// TwinCAT 3 PLC project Untitled1
// ProgramVersion: 3.1.4022.7
// libraries:
//   Tc2_MC2, * (Beckhoff Automation GmbH)
//   Tc2_MC2_Camming, * (Beckhoff Automation GmbH)
//   Tc2_Standard, * (Beckhoff Automation GmbH)
//   Tc2_System, * (Beckhoff Automation GmbH)
//   Tc3_Module, * (Beckhoff Automation GmbH)
// project tree:
//   DUTs/ ST_AxisIN.TcDUT, ST_AxisInterface.TcDUT, ST_AxisOUT.TcDUT
//   GVLs/ GVL_Servo.TcGVL
//   / PlcTask.TcTTO
//   POUs/ FB_Servo.TcPOU, MAIN.TcPOU, PRG_Camming.TcPOU
// real-time tasks:
//   TASK PlcTask: cycle T#10ms, priority 20, ADS port 350
// motion (NC):
//   TASK NC-Task 1 SAF: cycle T#2ms, priority 4, ADS port 501
//   TASK NC-Task 1 SVB: cycle T#10ms, priority 8, ADS port 511
//   AXIS Axis 3 (id 3)
//     Dynamic: Acceleration=12830, Deceleration=12830, Jerk=38490
//     Velo: RefSearch=85, RefSync=85, SlowManual=427, FastManual=2566, Fast=8553, Maximum=8553
//     OtherSettings: AllowMotionCmdToSlave=true
//     encoder EncType=8
//       EncPara: ScaleFactorNumerator=100, ScaleFactorDenominator=1048576, MaxCount=#xffffffff
//     drive DrvType=9
//       DrvPara: MaxCount=#xffffffff, DriveControlDWord=#x00030100
//         Analog: VeloReferenz=9408, ScaleFactorActTorque=0.1
//         TimeComp: TaskDelayCycles=1
//     controller CtrType=1
//       CtrPara: PriorControlFactor=1
//         Observer: BandWidth=20
//   AXIS Axis 4 (id 4)
//     Dynamic: Acceleration=12632, Deceleration=12632, Jerk=37898
//     Velo: RefSearch=84, RefSync=84, SlowManual=421, FastManual=2526, Fast=8421, Maximum=8421
//     OtherSettings: AllowMotionCmdToSlave=true
//     encoder EncType=8
//       EncPara: ScaleFactorNumerator=100, ScaleFactorDenominator=1048576, MaxCount=#xffffffff
//     drive DrvType=9
//       DrvPara: MaxCount=#xffffffff, DriveControlDWord=#x00030100
//         Analog: VeloReferenz=9264, ScaleFactorActTorque=0.1
//         TimeComp: TaskDelayCycles=1
//     controller CtrType=1
//       CtrPara: PriorControlFactor=1
//         Observer: BandWidth=20
// I/O:
//   DEVICE Device 1 (EtherCAT), AmsNetId 192.168.2.60.2.1
//     Term 1 (EK1200) [EK1200-5000 EtherCAT Power supply (2A E-Bus)]
//       Term 2 (EL1004) [EL1004 4Ch. Dig. Input 24V, 3ms]
//       Term 3 (EL2004) [EL2004 4Ch. Dig. Output 24V, 0.5A]
//       Term 4 (EL3062) [EL3062 2Ch. Ana. Input 0-10V]
//       Term 5 (EL4002) [EL4002 2Ch. Ana. Output 0-10V, 12bit]
//       Term 6 (EK1110) [EK1110 EtherCAT extension]
//     Drive 7 (AX5203-0000-0203) [AX5203-0000-0203 EtherCAT Drive (SoE, 2 Ch.)]
//   DEVICE Device 4 (USB)
//     Box 1 (CX2100 Power Supply)
//   DEVICE Device 5 (NOV-DP-RAM)
// variable links:
//   NC-Task 1 SAF/Axes/Axis 3 <-> Device 1 (EtherCAT)/Drive 7 (AX5203-0000-0203)
//     Drive/Inputs/In/nDataIn1 <-> AT 1/Following distance
//     Drive/Inputs/In/nDcOutputTime <-> InfoData/DcOutputShift
//     Drive/Inputs/In/nState1 <-> AT 1/Drive status word @bit 8
//     Drive/Inputs/In/nState2 <-> AT 1/Drive status word
//     Drive/Inputs/In/nState4 @bit 1 <-> WcState/InputToggle
//     Drive/Inputs/In/nState4 <-> WcState/WcState
//     Drive/Outputs/Out/nCtrl1 <-> MDT 1/Master control word @bit 8
//     Drive/Outputs/Out/nDataOut1 <-> MDT 1/Position command value
//     Enc/Inputs/In/nDataIn1 <-> AT 1/Position feedback 1 value
//     Enc/Inputs/In/nDcInputTime <-> InfoData/DcInputShift
//     Enc/Inputs/In/nState4 @bit 1 <-> WcState/InputToggle
//     Enc/Inputs/In/nState4 <-> WcState/WcState
//   NC-Task 1 SAF/Axes/Axis 4 <-> Device 1 (EtherCAT)/Drive 7 (AX5203-0000-0203)
//     Drive/Inputs/In/nDataIn1 <-> AT 2/Following distance
//     Drive/Inputs/In/nDcOutputTime <-> InfoData/DcOutputShift
//     Drive/Inputs/In/nState1 <-> AT 2/Drive status word @bit 8
//     Drive/Inputs/In/nState2 <-> AT 2/Drive status word
//     Drive/Inputs/In/nState4 @bit 1 <-> WcState/InputToggle
//     Drive/Inputs/In/nState4 <-> WcState/WcState
//     Drive/Outputs/Out/nCtrl1 <-> MDT 2/Master control word @bit 8
//     Drive/Outputs/Out/nDataOut1 <-> MDT 2/Position command value
//     Enc/Inputs/In/nDataIn1 <-> AT 2/Position feedback 1 value
//     Enc/Inputs/In/nDcInputTime <-> InfoData/DcInputShift
//     Enc/Inputs/In/nState4 @bit 1 <-> WcState/InputToggle
//     Enc/Inputs/In/nState4 <-> WcState/WcState
//   Untitled1/Untitled1 Instance <-> NC-Task 1 SAF/Axes/Axis 3
//     PlcTask Inputs/GVL_Servo.Axis1.NcToPlc <-> Outputs/ToPlc
//     PlcTask Outputs/GVL_Servo.Axis1.PlcToNc <-> Inputs/FromPlc
//   Untitled1/Untitled1 Instance <-> NC-Task 1 SAF/Axes/Axis 4
//     PlcTask Inputs/GVL_Servo.Axis2.NcToPlc <-> Outputs/ToPlc
//     PlcTask Outputs/GVL_Servo.Axis2.PlcToNc <-> Inputs/FromPlc

CONFIGURATION Untitled1
    RESOURCE PLC ON TwinCAT3
        TASK PlcTask(INTERVAL := T#10ms, PRIORITY := 20);
        PROGRAM MAIN WITH PlcTask : MAIN;
    END_RESOURCE
END_CONFIGURATION

// ---- DUTs/ST_AxisIN.TcDUT
TYPE ST_AxisIN :
STRUCT
	

bPower			:	BOOL;
nOverride		:	INT;

bAbs			:	BOOL;
fVelocity		:	LREAL;
fPos			:	LREAL;
            	
bCamIN			:	BOOL;
nCamTableID		:	UDINT;
bCamOUT			:	BOOL;
            	
bStop			:	BOOL;
            	
bReset			:	BOOL;
            	
bRead			:	BOOL;
            	
bWrite			:	BOOL;
nCamTableIdWr	:	UDINT;

END_STRUCT
END_TYPE

// ---- DUTs/ST_AxisInterface.TcDUT
TYPE ST_AxisInterface :
STRUCT
	
IN	:	ST_AxisIN;

OUT	:	ST_AxisOUT;

END_STRUCT
END_TYPE

// ---- DUTs/ST_AxisOUT.TcDUT
TYPE ST_AxisOUT :
STRUCT
	
bPowerEnabled	:	BOOL;
bPowerErr		:	BOOL;

bAbsDone		:	BOOL;
bAbsBusy		:	BOOL;
bAbsErr			:	BOOL;

bCamINDone		:	BOOL;

bCamOUTDone		:	BOOL;

bStopDone		:	BOOL;
bStopActive		:	BOOL;

bResetDone		:	BOOL;

bReadDone		:	BOOL;
bReadBusy		:	BOOL;
bReadErr		:	BOOL;

bWriteDone		:	BOOL;
bWriteBusy		:	BOOL;
bWriteErr		:	BOOL;

nCamTableIdWR	: UDINT;


END_STRUCT
END_TYPE

// ---- GVLs/GVL_Servo.TcGVL
VAR_GLOBAL
	
Axis1			:	AXIS_REF;
Axis2			:	AXIS_REF;

CAMTABLE		:	MC_CAM_REF;

AxisInterface1	:	ST_AxisInterface;

FB_Servo1		: FB_Servo;	


FB_Servo2		: FB_Servo;
AxisInterface2	: ST_AxisInterface;

MotionFunction	:	ARRAY [1..7] OF MC_MotionFunctionPoint;

arrSlavePos		: ARRAY[1..7]OF LREAL;
arrMasterPos	: ARRAY[1..7]OF LREAL;
	
END_VAR

// ---- POUs/MAIN.TcPOU
PROGRAM MAIN
VAR
END_VAR

PRG_Camming();
FB_Servo1(CAMTABLE:=CAMTABLE , Axis:=Axis1 , Slave:=Axis2 , stAxisInterface:=AxisInterface1 );
FB_Servo2(CAMTABLE:=CAMTABLE , Axis:=Axis2 , Slave:=Axis1 , stAxisInterface:=AxisInterface2 );

END_PROGRAM

// ---- POUs/PRG_Camming.TcPOU
PROGRAM PRG_Camming
VAR_INPUT
END_VAR
VAR_OUTPUT
END_VAR
VAR
	nState: INT;
	bExecute: BOOL;
	bWriteDoneButton: BOOL;
	ResetButton: BOOL;
END_VAR


MotionFunction[1].FunctionType	:=	MOTIONFUNCTYPE_SINUSLINIE;
MotionFunction[2].FunctionType	:=	MOTIONFUNCTYPE_SINUSLINIE;
MotionFunction[3].FunctionType	:=	MOTIONFUNCTYPE_SINUSLINIE;
MotionFunction[4].FunctionType	:=	MOTIONFUNCTYPE_SINUSLINIE;
MotionFunction[5].FunctionType	:=	MOTIONFUNCTYPE_SINUSLINIE;
MotionFunction[6].FunctionType	:=	MOTIONFUNCTYPE_SINUSLINIE;


CAMTABLE.TableType	:= MC_TABLETYPE_MOTIONFUNCTION;
CAMTABLE.pArray		:= ADR(MotionFunction);
CAMTABLE.ArraySize	:= SIZEOF(MotionFunction);
CAMTABLE.NoOfColumns:= 1;
CAMTABLE.NoOfRows	:= SIZEOF(MotionFunction)/SIZEOF(MotionFunction[1]);


AxisInterface1.IN.bPower	:=	TRUE;
AxisInterface1.IN.nOverride	:=	100;

AxisInterface2.IN.bPower	:=	TRUE;
AxisInterface2.IN.nOverride	:=	100;



CASE nState	OF
	
	0:
		IF bExecute	
		AND AxisInterface1.OUT.bPowerEnabled 
		AND AxisInterface2.OUT.bPowerEnabled	THEN
			Axisinterface1.IN.bStop		:=	FALSE;
			Axisinterface2.IN.bStop		:=	FALSE;
			
			IF NOT AxisInterface1.OUT.bStopActive AND NOT AxisInterface2.OUT.bStopActive THEN
							nState:=5;
			END_IF
			
		END_IF
		
		
	5:
		AxisInterface1.IN.bCamIN	:=TRUE;
		AxisInterface1.IN.nCamTableID	:=	1;
		
		IF AxisInterface1.OUT.bCamINDone	THEN			
			AxisInterface1.IN.bCamIN	:=FALSE;
			nState						:=	10;			
		END_IF
	
	10:
			

			IF AxisInterface1.OUT.bPowerEnabled 
			AND AxisInterface2.OUT.bPowerEnabled	THEN
			
	
			
			AxisInterface1.IN.fPos		:=	18000;
			AxisInterface1.IN.fVelocity	:=	1500;
		
			AxisInterface1.IN.bAbs		:=	TRUE;			
			nstate	:=	20;
			
			
		
		ELSIF Axisinterface1.OUT.bAbsErr	THEN
			nState	:=	999;
		END_IF
		
	
			
			20:	
		IF AxisInterface1.OUT.bAbsBusy
		AND NOT AxisInterface1.OUT.bAbsErr	THEN
			
			nState	:=	30;
			
			ELSIF Axisinterface1.OUT.bAbsErr	THEN
				nState	:=	999;
			END_IF
			
	
	30:
		IF AxisInterface1.OUT.bAbsDone
		AND NOT AxisInterface1.OUT.bAbsErr	THEN
		
		AxisInterface1.IN.bAbs		:=	FALSE;
		AxisInterface1.IN.bCamOUT	:=	TRUE;
		AxisInterface1.IN.bCamIN	:=FALSE;

		nState	:=	31;
		
			
		ELSIF Axisinterface1.OUT.bAbsErr	THEN
	//	nState	:=	999;
			
		END_IF
		
		31:
			IF AxisInterface1.OUT.bCamOUTDone	THEN
				nState	:=	32;
				AxisInterface1.IN.bCamOUT	:=	FALSE;
			END_IF
		
	32:
		AxisInterface1.IN.bRead	:=	TRUE;
		AxisInterface1.IN.nCamTableIdWr	:=	1;

			IF AxisInterface1.OUT.bReadDone THEN
				nState	:=40;
				AxisInterface1.IN.bRead	:= FALSE;		
			END_IF
		
		
	40:
	
		MotionFunction[1].SlavePos	:= arrSlavePos[1];
		MotionFunction[2].SlavePos	:= arrSlavePos[2];
		MotionFunction[3].SlavePos	:= arrSlavePos[3];
		MotionFunction[4].SlavePos	:= arrSlavePos[4];
		MotionFunction[5].SlavePos	:= arrSlavePos[5];
		MotionFunction[6].SlavePos	:= arrSlavePos[6];
		MotionFunction[7].SlavePos	:= arrSlavePos[7];
		
		MotionFunction[1].MasterPos	:= 0;
		MotionFunction[2].MasterPos	:= 60;
		MotionFunction[3].MasterPos	:= 120;
		MotionFunction[4].MasterPos	:= 180;
		MotionFunction[5].MasterPos	:= 240;
		MotionFunction[6].MasterPos	:= 300;
		MotionFunction[7].MasterPos	:= 360;
		
	
		
		
		
AxisInterface1.IN.bWrite	:=	bWriteDoneButton;
		
		IF AxisInterface1.OUT.bWriteDone	 THEN
			AxisInterface1.IN.bWrite	:= FALSE;
			nState					:= 50;		
		END_IF
	
	50:
		
		IF AxisInterface1.OUT.bPowerEnabled 
		AND AxisInterface1.OUT.bPowerEnabled
		AND NOT AxisInterface1.OUT.bAbsErr	THEN
		
			AxisInterface1.IN.fPos		:=	0;
			AxisInterface1.IN.fVelocity	:=	2000;
			AxisInterface1.IN.bAbs		:=	TRUE;
			
			nState						:=	60;
			
	
		ELSIF Axisinterface1.OUT.bAbsErr	THEN
			nState	:=	999;
		END_IF
	
	60:
	
		IF AxisInterface1.OUT.bAbsBusy
		AND NOT AxisInterface1.OUT.bAbsErr	THEN
			
			nState	:=	70;
			AxisInterface1.IN.bAbs		:=	FALSE;
			
		ELSIF Axisinterface1.OUT.bAbsErr	THEN
			nState	:=	999;
		END_IF
			

	70:
		
		IF AxisInterface1.OUT.babsdone
		AND NOT AxisInterface1.OUT.bAbsErr	THEN
		
			nState	:=	0;

			
		ELSIF Axisinterface1.OUT.bAbsErr	THEN
				nState	:=	999;
		END_IF
		
END_CASE

IF NOT bExecute THEN
	
	AxisInterface1.IN.bStop	:=	TRUE;
	AxisInterface2.IN.bStop	:=	TRUE;

	AxisInterface1.IN.bAbs	:=	FALSE;

		
END_IF
	
	
IF ResetButton THEN


	AxisInterface1.IN.bReset	:=	TRUE;	
	
	IF AxisInterface1.OUT.bResetDone	THEN
		nState	:=	0;
		bExecute	:=	FALSE;
	END_IF

END_IF

END_PROGRAM

// ---- POUs/FB_Servo.TcPOU
FUNCTION_BLOCK FB_Servo
VAR_INPUT
	CAMTABLE		: MC_CAM_REF;
END_VAR
VAR_OUTPUT
END_VAR
VAR
	McPower: MC_Power;
	McReset: MC_Reset;
	McMoveAbs: MC_MoveAbsolute;
	McCamIN: MC_CamIn_V2;
	McCamOUT: MC_CamOut;
	McStop: MC_Stop;
	McWrite: MC_WriteMotionFunction;
	McRead: MC_ReadMotionFunction;
END_VAR
VAR_IN_OUT
	Axis			:	AXIS_REF;
	Slave			:	AXIS_REf;
	stAxisInterface	:	ST_AxisInterface;
END_VAR

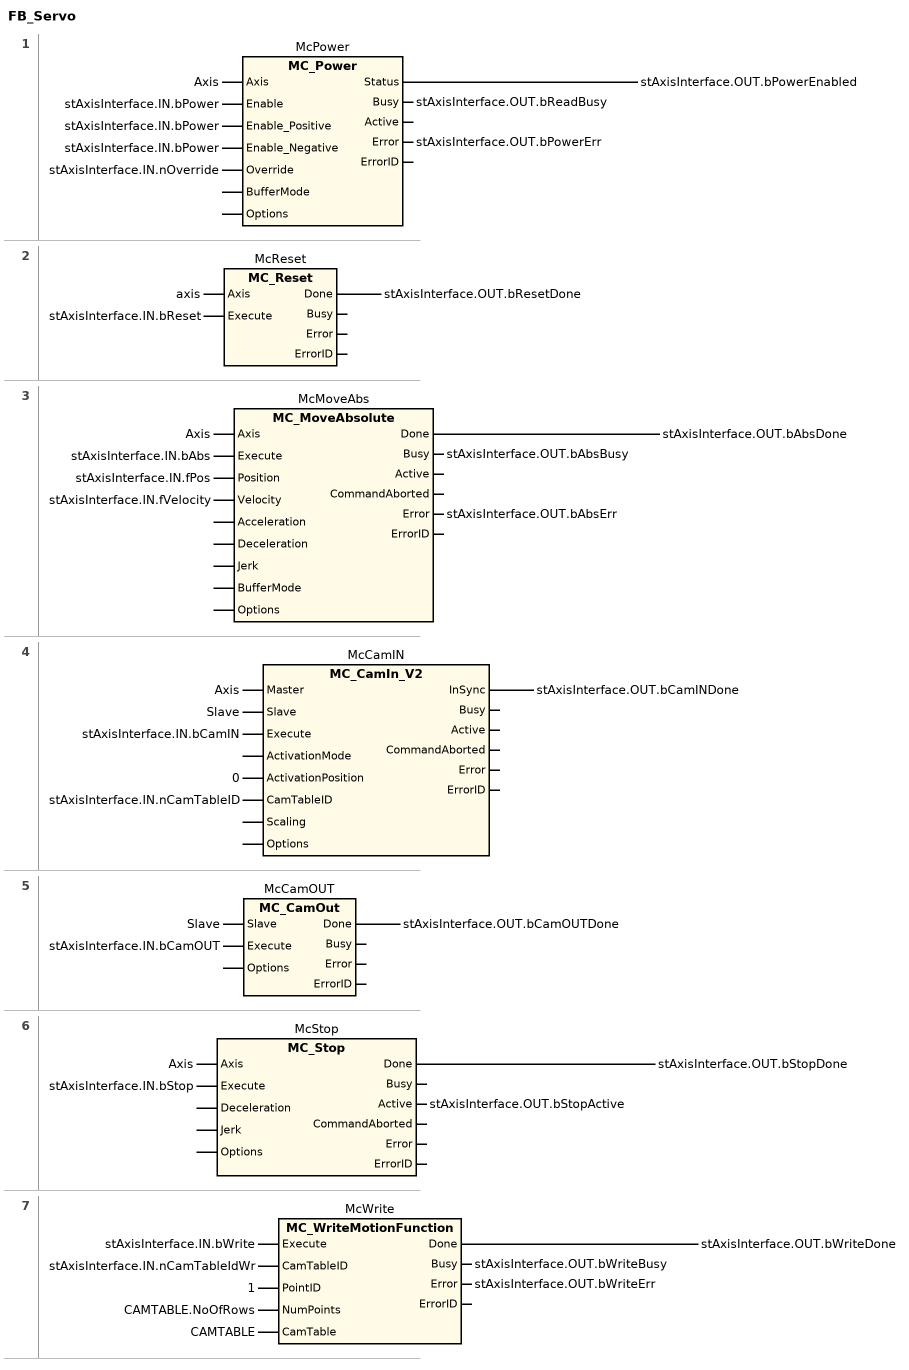
// NETWORK 1
McPower(
    Axis := Axis,
    Enable := stAxisInterface.IN.bPower,
    Enable_Positive := stAxisInterface.IN.bPower,
    Enable_Negative := stAxisInterface.IN.bPower,
    Override := stAxisInterface.IN.nOverride,
    Busy => stAxisInterface.OUT.bReadBusy,
    Error => stAxisInterface.OUT.bPowerErr); // MC_Power
stAxisInterface.OUT.bPowerEnabled := McPower.Status;

// NETWORK 2
McReset(Axis := axis, Execute := stAxisInterface.IN.bReset); // MC_Reset
stAxisInterface.OUT.bResetDone := McReset.Done;

// NETWORK 3
McMoveAbs(
    Axis := Axis,
    Execute := stAxisInterface.IN.bAbs,
    Position := stAxisInterface.IN.fPos,
    Velocity := stAxisInterface.IN.fVelocity,
    Busy => stAxisInterface.OUT.bAbsBusy,
    Error => stAxisInterface.OUT.bAbsErr); // MC_MoveAbsolute
stAxisInterface.OUT.bAbsDone := McMoveAbs.Done;

// NETWORK 4
McCamIN(
    Master := Axis,
    Slave := Slave,
    Execute := stAxisInterface.IN.bCamIN,
    ActivationPosition := 0,
    CamTableID := stAxisInterface.IN.nCamTableID); // MC_CamIn_V2
stAxisInterface.OUT.bCamINDone := McCamIN.InSync;

// NETWORK 5
McCamOUT(Slave := Slave, Execute := stAxisInterface.IN.bCamOUT); // MC_CamOut
stAxisInterface.OUT.bCamOUTDone := McCamOUT.Done;

// NETWORK 6
McStop(Axis := Axis, Execute := stAxisInterface.IN.bStop, Active => stAxisInterface.OUT.bStopActive); // MC_Stop
stAxisInterface.OUT.bStopDone := McStop.Done;

// NETWORK 7
McWrite(
    Execute := stAxisInterface.IN.bWrite,
    CamTableID := stAxisInterface.IN.nCamTableIdWr,
    PointID := 1,
    NumPoints := CAMTABLE.NoOfRows,
    CamTable := CAMTABLE,
    Busy => stAxisInterface.OUT.bWriteBusy,
    Error => stAxisInterface.OUT.bWriteErr); // MC_WriteMotionFunction
stAxisInterface.OUT.bWriteDone := McWrite.Done;

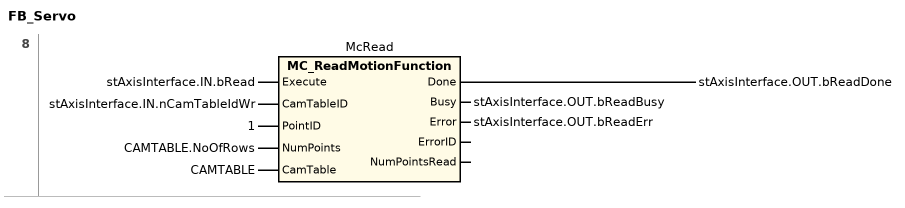
// NETWORK 8
McRead(
    Execute := stAxisInterface.IN.bRead,
    CamTableID := stAxisInterface.IN.nCamTableIdWr,
    PointID := 1,
    NumPoints := CAMTABLE.NoOfRows,
    CamTable := CAMTABLE,
    Busy => stAxisInterface.OUT.bReadBusy,
    Error => stAxisInterface.OUT.bReadErr); // MC_ReadMotionFunction
stAxisInterface.OUT.bReadDone := McRead.Done;

END_FUNCTION_BLOCK
